{attribute 'GeneratedUsingTerminal: EL3632-0000-0016'}
{attribute addProperty BoxType "EL3632-0000-0016"}
{attribute addProperty Id "Ch2_ValueAT %I*INT2"}
{attribute addProperty CRC "2674427622"}
{attribute addProperty Size "2"}
TYPE Ch2_Sample_9F6886E6 :
STRUCT
	{attribute addProperty Name "Ch2_Value"}
	Ch2_Value AT %I* : INT;
END_STRUCT
END_TYPE

(* stored: Version 1.2.0.0, ProductVersion 3.1.4024.9
   DUT Ch2_Sample_9F6886E6: Id {9df6a4d9-3ce1-4ff0-ab4c-09ee41f51569} *)
